(*********************************** G.D S.p.A. - Technical Department ***********************************
============= PROGRAM INFO ============
FOLDER:             TBD
MACHINES INVOLVED:  TBD 

============= DESCRIPTION =============
Machine declaration

============= REVISIONS ===============
Date		Version	 	Author      	Description             
----------	-------		------------  	--------------------------------------------
2019/03/27 	0000.00	 	CEC 			Creation of the PRG

**********************************************************************************************************)

TYPE csp_customerInterfaces_casePackerLabels :
STRUCT
	
	Consumed:						DINT;				(*$H_R desc := Real time total material consumption for this order; $*)
															
END_STRUCT
END_TYPE

(* stored: Version 1.1.0.1, ProductVersion 3.1.4024.3
   DUT csp_customerInterfaces_casePackerLabels: Id {61c054b4-c54d-445a-98f3-003ea8a07024} *)
